PROGRAM PRG_TEST
VAR
	_problem1Test : Problem1Test;
END_VAR

TcUnit.RUN();

END_PROGRAM

(* stored: Version 1.1.0.1, ProductVersion 3.1.4024.9
   POU PRG_TEST: Id {dcb4004d-c8d2-4d22-a248-44f6a6dc5a3f}, SpecialFunc None *)
